// TIA Portal project "Trabajo" (V15)

(* hardware
DEVICE "S7-1200 station_1"  S7-1200 Station
   slot 0: "Rack_0"  S7-1200 Rack  Rack  V1.0
   slot 1: "PLC_1"  CPU 1215C AC/DC/Rly  6ES7 215-1BG40-0XB0  V4.2
*)

// ===== PLC "PLC_1"  CPU 1215C AC/DC/Rly =====

VAR_GLOBAL   // PLC tag table "Tabla de variables estándar"
   "Marcha" AT %I0.0 : Bool;
   "STOP" AT %I0.1 : Bool;
   "Automático" AT %I0.2 : Bool;
   "C1 Extendido" AT %I0.3 : Bool;
   "C1 Recogido" AT %I0.4 : Bool;
   "C2 Extendido" AT %I0.5 : Bool;
   "C2 Recogido" AT %I0.6 : Bool;
   "C3 Extendido" AT %I0.7 : Bool;
   "C3 Recogido" AT %I1.0 : Bool;
   "Alimentación" AT %I1.1 : Bool;
   "Pieza Mesa" AT %I1.2 : Bool;
   "Marcha 0" AT %M30.0 : Bool;
   "Marcha 1" AT %M30.1 : Bool;
   "Marcha 2" AT %M30.2 : Bool;
   "Marcha 3" AT %M30.3 : Bool;
   "Marcha 4" AT %M30.4 : Bool;
   "Marcha 5" AT %M30.5 : Bool;
   "Marcha 6" AT %M30.6 : Bool;
   "Marcha 7" AT %M30.7 : Bool;
   "Marcha 8" AT %M31.0 : Bool;
   "Marcha 9" AT %M31.1 : Bool;
   "Marcha 10" AT %M31.2 : Bool;
   "Marcha 11" AT %M31.3 : Bool;
   "Marcha 12" AT %M31.4 : Bool;
   "STOP 0" AT %M3.0 : Bool;
   "STOP 1" AT %M3.1 : Bool;
   "STOP 2" AT %M3.2 : Bool;
   "STOP 3" AT %M3.3 : Bool;
   "STOP 4" AT %M3.4 : Bool;
   "STOP 5" AT %M3.5 : Bool;
   "C1 SET" AT %Q0.0 : Bool;
   "C1 RESET" AT %Q0.1 : Bool;
   "C2 SET" AT %Q0.2 : Bool;
   "C2 RESET" AT %Q0.3 : Bool;
   "C3 SET" AT %Q0.4 : Bool;
   "Cinta ON" AT %Q0.5 : Bool;
   "Cinta INVERSA" AT %Q0.6 : Bool;
   "NumPiezas" AT %MW50 : Int;
   "Marcha 13" AT %M31.5 : Bool;
   "Marcha 14" AT %M31.6 : Bool;
   "Tag_2" AT %MB3 : Byte;
   "Tag_3" AT %MW30 : Int;
   "Tag_1" AT %MW100 : Int;
END_VAR

// folder: System blocks/Program resources

DATA_BLOCK "T1"   // DB1
{ S7_Optimized_Access := 'TRUE' }
AUTHOR : Simatic
FAMILY : IEC
NAME : IEC_TMR
VERSION : 1.0
// stored: InstanceOfName IEC_TIMER
"IEC_TIMER"
BEGIN
END_DATA_BLOCK

DATA_BLOCK "T2"   // DB2
{ S7_Optimized_Access := 'TRUE' }
AUTHOR : Simatic
FAMILY : IEC
NAME : IEC_TMR
VERSION : 1.0
// stored: InstanceOfName IEC_TIMER
"IEC_TIMER"
BEGIN
END_DATA_BLOCK

DATA_BLOCK "T3"   // DB3
{ S7_Optimized_Access := 'TRUE' }
AUTHOR : Simatic
FAMILY : IEC
NAME : IEC_TMR
VERSION : 1.0
// stored: InstanceOfName IEC_TIMER
"IEC_TIMER"
BEGIN
END_DATA_BLOCK

DATA_BLOCK "Contador"   // DB4
{ S7_Optimized_Access := 'TRUE' }
AUTHOR : Simatic
FAMILY : IEC
NAME : CNTR
VERSION : 1.0
// stored: InstanceOfName IEC_COUNTER
"IEC_COUNTER"
BEGIN
END_DATA_BLOCK

// folder: (top level)

FUNCTION "F_Marcha" : Void   // FC1, LAD
{ S7_Optimized_Access := 'TRUE' }
VERSION : 0.1
BEGIN

REGION Network 1: Etapa 0
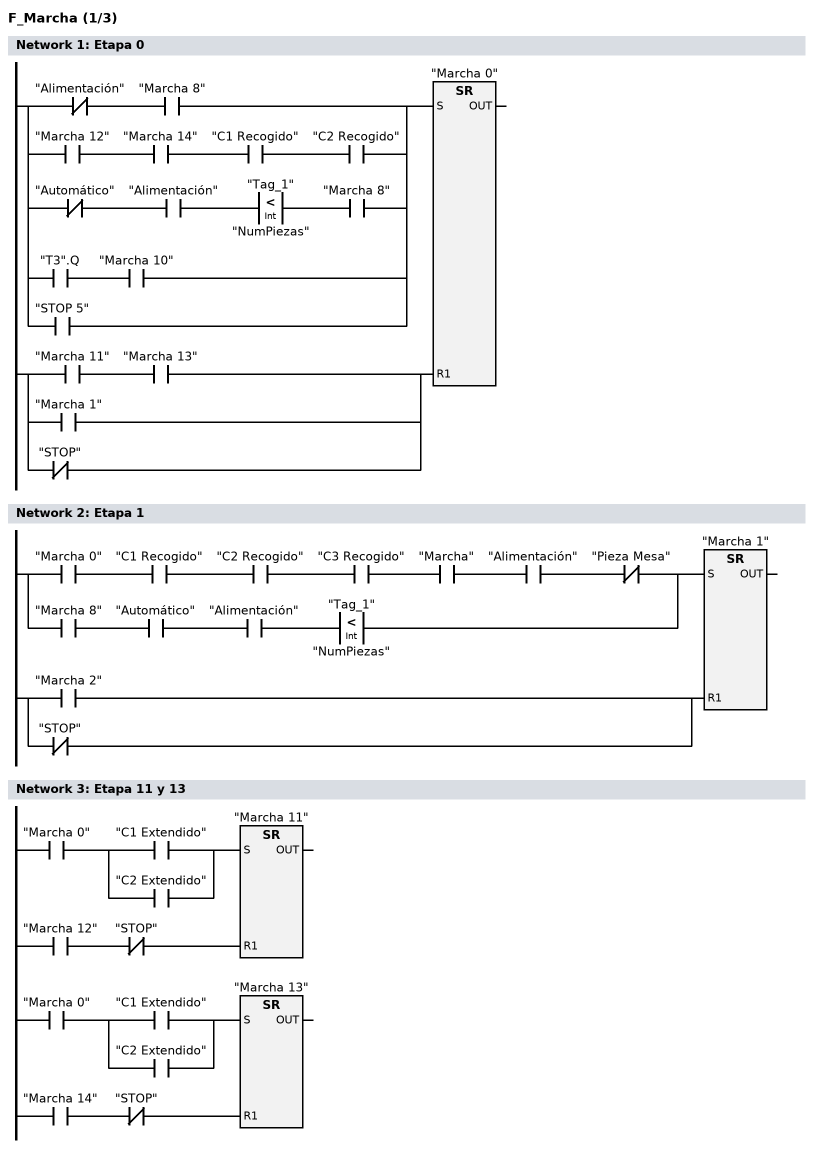
   RUNG wire#powerrail
      I_Contact( "Alimentación" )
      Contact( "Marcha 8" )
      wire#w1
      S_SR(operand := "Marcha 0", r1 := wire#w2)
   END_RUNG
   RUNG wire#powerrail
      Contact( "Marcha 12" )
      Contact( "Marcha 14" )
      Contact( "C1 Recogido" )
      Contact( "C2 Recogido" )
   END_RUNG wire#w1
   RUNG wire#powerrail
      I_Contact( "Automático" )
      Contact( "Alimentación" )
      { S7_Templates := "SrcType := Int" } LT_Contact(in1 := "Tag_1", in2 := "NumPiezas")
      Contact( "Marcha 8" )
   END_RUNG wire#w1
   RUNG wire#powerrail
      Contact( "T3".Q )
      Contact( "Marcha 10" )
   END_RUNG wire#w1
   RUNG wire#powerrail
      Contact( "STOP 5" )
   END_RUNG wire#w1
   RUNG wire#powerrail
      Contact( "Marcha 11" )
      Contact( "Marcha 13" )
   END_RUNG wire#w2
   RUNG wire#powerrail
      Contact( "Marcha 1" )
   END_RUNG wire#w2
   RUNG wire#powerrail
      I_Contact( "STOP" )
   END_RUNG wire#w2
   // the same network as SCL:
   IF (NOT "Alimentación" AND "Marcha 8") OR ("Marcha 12" AND "Marcha 14" AND "C1 Recogido" AND "C2 Recogido") OR (NOT "Automático" AND "Alimentación" AND ("Tag_1" < "NumPiezas") AND "Marcha 8") OR ("T3".Q AND "Marcha 10") OR "STOP 5" THEN
       "Marcha 0" := TRUE;   // SR flip-flop
   END_IF;
   IF ("Marcha 11" AND "Marcha 13") OR "Marcha 1" OR NOT "STOP" THEN "Marcha 0" := FALSE; END_IF;
END_REGION

REGION Network 2: Etapa 1
   RUNG wire#powerrail
      Contact( "Marcha 0" )
      Contact( "C1 Recogido" )
      Contact( "C2 Recogido" )
      Contact( "C3 Recogido" )
      Contact( "Marcha" )
      Contact( "Alimentación" )
      I_Contact( "Pieza Mesa" )
      wire#w1
      S_SR(operand := "Marcha 1", r1 := wire#w2)
   END_RUNG
   RUNG wire#powerrail
      Contact( "Marcha 8" )
      Contact( "Automático" )
      Contact( "Alimentación" )
      { S7_Templates := "SrcType := Int" } LT_Contact(in1 := "Tag_1", in2 := "NumPiezas")
   END_RUNG wire#w1
   RUNG wire#powerrail
      Contact( "Marcha 2" )
   END_RUNG wire#w2
   RUNG wire#powerrail
      I_Contact( "STOP" )
   END_RUNG wire#w2
   // the same network as SCL:
   IF ("Marcha 0" AND "C1 Recogido" AND "C2 Recogido" AND "C3 Recogido" AND "Marcha" AND "Alimentación" AND NOT "Pieza Mesa") OR ("Marcha 8" AND "Automático" AND "Alimentación" AND ("Tag_1" < "NumPiezas")) THEN
       "Marcha 1" := TRUE;   // SR flip-flop
   END_IF;
   IF "Marcha 2" OR NOT "STOP" THEN "Marcha 1" := FALSE; END_IF;
END_REGION

REGION Network 3: Etapa 11 y 13
   RUNG wire#powerrail
      Contact( "Marcha 0" )
      wire#w1
      Contact( "C1 Extendido" )
      wire#w2
      S_SR(operand := "Marcha 11", r1 := wire#w3)
   END_RUNG
   RUNG wire#w1
      Contact( "C2 Extendido" )
   END_RUNG wire#w2
   RUNG wire#powerrail
      Contact( "Marcha 12" )
      I_Contact( "STOP" )
   END_RUNG wire#w3
   RUNG wire#powerrail
      Contact( "Marcha 0" )
      wire#w4
      Contact( "C1 Extendido" )
      wire#w5
      S_SR(operand := "Marcha 13", r1 := wire#w6)
   END_RUNG
   RUNG wire#w4
      Contact( "C2 Extendido" )
   END_RUNG wire#w5
   RUNG wire#powerrail
      Contact( "Marcha 14" )
      I_Contact( "STOP" )
   END_RUNG wire#w6
   // the same network as SCL:
   IF "Marcha 0" AND ("C1 Extendido" OR "C2 Extendido") THEN
       "Marcha 11" := TRUE;   // SR flip-flop
   END_IF;
   IF "Marcha 12" AND NOT "STOP" THEN "Marcha 11" := FALSE; END_IF;
   IF "Marcha 0" AND ("C1 Extendido" OR "C2 Extendido") THEN
       "Marcha 13" := TRUE;   // SR flip-flop
   END_IF;
   IF "Marcha 14" AND NOT "STOP" THEN "Marcha 13" := FALSE; END_IF;
END_REGION

REGION Network 4: Etapa 12 y 14
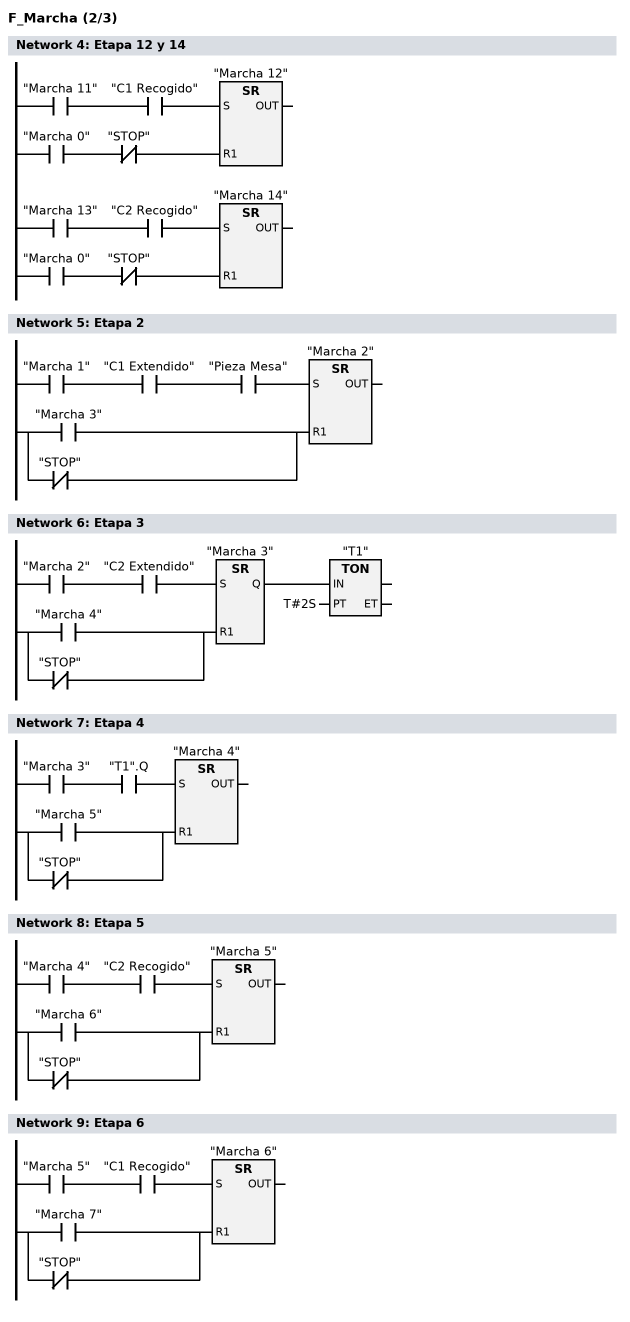
   RUNG wire#powerrail
      Contact( "Marcha 11" )
      Contact( "C1 Recogido" )
      S_SR(operand := "Marcha 12", r1 := wire#w1)
   END_RUNG
   RUNG wire#powerrail
      Contact( "Marcha 0" )
      I_Contact( "STOP" )
   END_RUNG wire#w1
   RUNG wire#powerrail
      Contact( "Marcha 13" )
      Contact( "C2 Recogido" )
      S_SR(operand := "Marcha 14", r1 := wire#w2)
   END_RUNG
   RUNG wire#powerrail
      Contact( "Marcha 0" )
      I_Contact( "STOP" )
   END_RUNG wire#w2
   // the same network as SCL:
   IF "Marcha 11" AND "C1 Recogido" THEN
       "Marcha 12" := TRUE;   // SR flip-flop
   END_IF;
   IF "Marcha 0" AND NOT "STOP" THEN "Marcha 12" := FALSE; END_IF;
   IF "Marcha 13" AND "C2 Recogido" THEN
       "Marcha 14" := TRUE;   // SR flip-flop
   END_IF;
   IF "Marcha 0" AND NOT "STOP" THEN "Marcha 14" := FALSE; END_IF;
END_REGION

REGION Network 5: Etapa 2
   RUNG wire#powerrail
      Contact( "Marcha 1" )
      Contact( "C1 Extendido" )
      Contact( "Pieza Mesa" )
      S_SR(operand := "Marcha 2", r1 := wire#w1)
   END_RUNG
   RUNG wire#powerrail
      Contact( "Marcha 3" )
   END_RUNG wire#w1
   RUNG wire#powerrail
      I_Contact( "STOP" )
   END_RUNG wire#w1
   // the same network as SCL:
   IF "Marcha 1" AND "C1 Extendido" AND "Pieza Mesa" THEN
       "Marcha 2" := TRUE;   // SR flip-flop
   END_IF;
   IF "Marcha 3" OR NOT "STOP" THEN "Marcha 2" := FALSE; END_IF;
END_REGION

REGION Network 6: Etapa 3
   IF "Marcha 2" AND "C2 Extendido" THEN
       "Marcha 3" := TRUE;   // SR flip-flop
   END_IF;
   IF "Marcha 4" OR NOT "STOP" THEN "Marcha 3" := FALSE; END_IF;
   "T1".TON(IN := "Marcha 3", PT := T#2S);
END_REGION

REGION Network 7: Etapa 4
   RUNG wire#powerrail
      Contact( "Marcha 3" )
      Contact( "T1".Q )
      S_SR(operand := "Marcha 4", r1 := wire#w1)
   END_RUNG
   RUNG wire#powerrail
      Contact( "Marcha 5" )
   END_RUNG wire#w1
   RUNG wire#powerrail
      I_Contact( "STOP" )
   END_RUNG wire#w1
   // the same network as SCL:
   IF "Marcha 3" AND "T1".Q THEN
       "Marcha 4" := TRUE;   // SR flip-flop
   END_IF;
   IF "Marcha 5" OR NOT "STOP" THEN "Marcha 4" := FALSE; END_IF;
END_REGION

REGION Network 8: Etapa 5
   RUNG wire#powerrail
      Contact( "Marcha 4" )
      Contact( "C2 Recogido" )
      S_SR(operand := "Marcha 5", r1 := wire#w1)
   END_RUNG
   RUNG wire#powerrail
      Contact( "Marcha 6" )
   END_RUNG wire#w1
   RUNG wire#powerrail
      I_Contact( "STOP" )
   END_RUNG wire#w1
   // the same network as SCL:
   IF "Marcha 4" AND "C2 Recogido" THEN
       "Marcha 5" := TRUE;   // SR flip-flop
   END_IF;
   IF "Marcha 6" OR NOT "STOP" THEN "Marcha 5" := FALSE; END_IF;
END_REGION

REGION Network 9: Etapa 6
   RUNG wire#powerrail
      Contact( "Marcha 5" )
      Contact( "C1 Recogido" )
      S_SR(operand := "Marcha 6", r1 := wire#w1)
   END_RUNG
   RUNG wire#powerrail
      Contact( "Marcha 7" )
   END_RUNG wire#w1
   RUNG wire#powerrail
      I_Contact( "STOP" )
   END_RUNG wire#w1
   // the same network as SCL:
   IF "Marcha 5" AND "C1 Recogido" THEN
       "Marcha 6" := TRUE;   // SR flip-flop
   END_IF;
   IF "Marcha 7" OR NOT "STOP" THEN "Marcha 6" := FALSE; END_IF;
END_REGION

REGION Network 10: Etapa 7
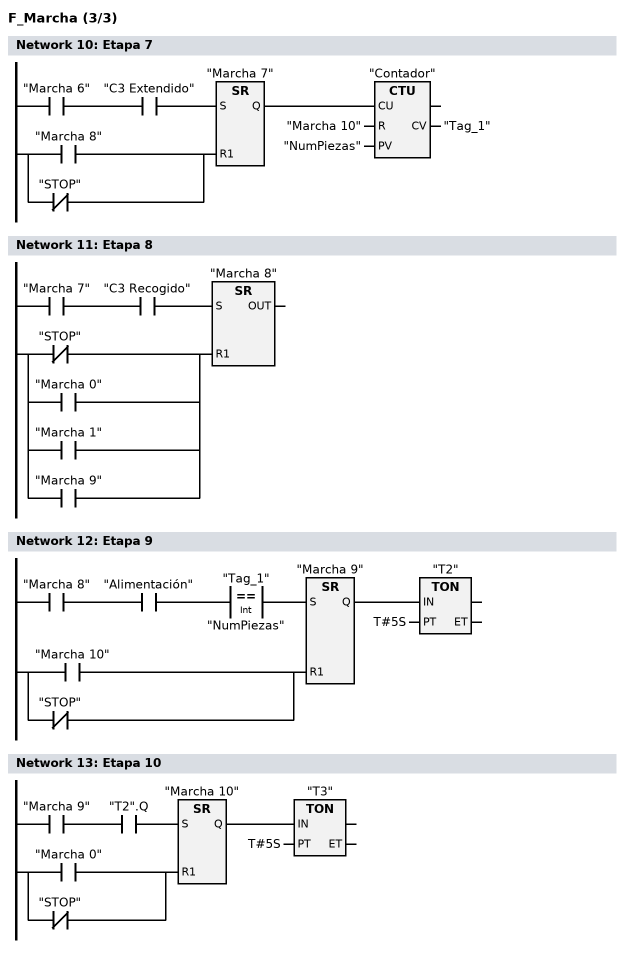
   IF "Marcha 6" AND "C3 Extendido" THEN
       "Marcha 7" := TRUE;   // SR flip-flop
   END_IF;
   IF "Marcha 8" OR NOT "STOP" THEN "Marcha 7" := FALSE; END_IF;
   "Contador".CTU(CU := "Marcha 7", R := "Marcha 10", PV := "NumPiezas", CV => "Tag_1");
END_REGION

REGION Network 11: Etapa 8
   RUNG wire#powerrail
      Contact( "Marcha 7" )
      Contact( "C3 Recogido" )
      S_SR(operand := "Marcha 8", r1 := wire#w1)
   END_RUNG
   RUNG wire#powerrail
      I_Contact( "STOP" )
   END_RUNG wire#w1
   RUNG wire#powerrail
      Contact( "Marcha 0" )
   END_RUNG wire#w1
   RUNG wire#powerrail
      Contact( "Marcha 1" )
   END_RUNG wire#w1
   RUNG wire#powerrail
      Contact( "Marcha 9" )
   END_RUNG wire#w1
   // the same network as SCL:
   IF "Marcha 7" AND "C3 Recogido" THEN
       "Marcha 8" := TRUE;   // SR flip-flop
   END_IF;
   IF NOT "STOP" OR "Marcha 0" OR "Marcha 1" OR "Marcha 9" THEN "Marcha 8" := FALSE; END_IF;
END_REGION

REGION Network 12: Etapa 9
   IF "Marcha 8" AND "Alimentación" AND ("Tag_1" = "NumPiezas") THEN
       "Marcha 9" := TRUE;   // SR flip-flop
   END_IF;
   IF "Marcha 10" OR NOT "STOP" THEN "Marcha 9" := FALSE; END_IF;
   "T2".TON(IN := "Marcha 9", PT := T#5S);
END_REGION

REGION Network 13: Etapa 10
   IF "Marcha 9" AND "T2".Q THEN
       "Marcha 10" := TRUE;   // SR flip-flop
   END_IF;
   IF "Marcha 0" OR NOT "STOP" THEN "Marcha 10" := FALSE; END_IF;
   "T3".TON(IN := "Marcha 10", PT := T#5S);
END_REGION
END_FUNCTION

FUNCTION "F_STOP" : Void   // FC2, LAD
{ S7_Optimized_Access := 'TRUE' }
VERSION : 0.1
BEGIN

REGION Network 1: Etapa 0
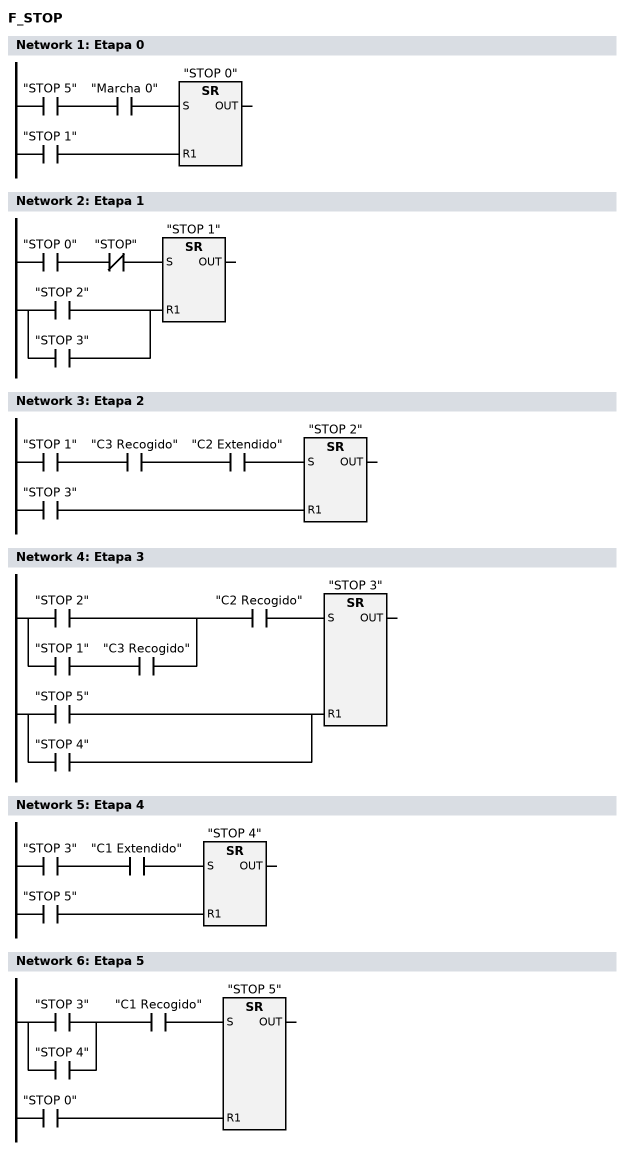
   RUNG wire#powerrail
      Contact( "STOP 5" )
      Contact( "Marcha 0" )
      S_SR(operand := "STOP 0", r1 := wire#w1)
   END_RUNG
   RUNG wire#powerrail
      Contact( "STOP 1" )
   END_RUNG wire#w1
   // the same network as SCL:
   IF "STOP 5" AND "Marcha 0" THEN
       "STOP 0" := TRUE;   // SR flip-flop
   END_IF;
   IF "STOP 1" THEN "STOP 0" := FALSE; END_IF;
END_REGION

REGION Network 2: Etapa 1
   RUNG wire#powerrail
      Contact( "STOP 0" )
      I_Contact( "STOP" )
      S_SR(operand := "STOP 1", r1 := wire#w1)
   END_RUNG
   RUNG wire#powerrail
      Contact( "STOP 2" )
   END_RUNG wire#w1
   RUNG wire#powerrail
      Contact( "STOP 3" )
   END_RUNG wire#w1
   // the same network as SCL:
   IF "STOP 0" AND NOT "STOP" THEN
       "STOP 1" := TRUE;   // SR flip-flop
   END_IF;
   IF "STOP 2" OR "STOP 3" THEN "STOP 1" := FALSE; END_IF;
END_REGION

REGION Network 3: Etapa 2
   RUNG wire#powerrail
      Contact( "STOP 1" )
      Contact( "C3 Recogido" )
      Contact( "C2 Extendido" )
      S_SR(operand := "STOP 2", r1 := wire#w1)
   END_RUNG
   RUNG wire#powerrail
      Contact( "STOP 3" )
   END_RUNG wire#w1
   // the same network as SCL:
   IF "STOP 1" AND "C3 Recogido" AND "C2 Extendido" THEN
       "STOP 2" := TRUE;   // SR flip-flop
   END_IF;
   IF "STOP 3" THEN "STOP 2" := FALSE; END_IF;
END_REGION

REGION Network 4: Etapa 3
   RUNG wire#powerrail
      Contact( "STOP 2" )
      wire#w1
      Contact( "C2 Recogido" )
      S_SR(operand := "STOP 3", r1 := wire#w2)
   END_RUNG
   RUNG wire#powerrail
      Contact( "STOP 1" )
      Contact( "C3 Recogido" )
   END_RUNG wire#w1
   RUNG wire#powerrail
      Contact( "STOP 5" )
   END_RUNG wire#w2
   RUNG wire#powerrail
      Contact( "STOP 4" )
   END_RUNG wire#w2
   // the same network as SCL:
   IF ("STOP 2" OR ("STOP 1" AND "C3 Recogido")) AND "C2 Recogido" THEN
       "STOP 3" := TRUE;   // SR flip-flop
   END_IF;
   IF "STOP 5" OR "STOP 4" THEN "STOP 3" := FALSE; END_IF;
END_REGION

REGION Network 5: Etapa 4
   RUNG wire#powerrail
      Contact( "STOP 3" )
      Contact( "C1 Extendido" )
      S_SR(operand := "STOP 4", r1 := wire#w1)
   END_RUNG
   RUNG wire#powerrail
      Contact( "STOP 5" )
   END_RUNG wire#w1
   // the same network as SCL:
   IF "STOP 3" AND "C1 Extendido" THEN
       "STOP 4" := TRUE;   // SR flip-flop
   END_IF;
   IF "STOP 5" THEN "STOP 4" := FALSE; END_IF;
END_REGION

REGION Network 6: Etapa 5
   RUNG wire#powerrail
      Contact( "STOP 3" )
      wire#w1
      Contact( "C1 Recogido" )
      S_SR(operand := "STOP 5", r1 := wire#w2)
   END_RUNG
   RUNG wire#powerrail
      Contact( "STOP 4" )
   END_RUNG wire#w1
   RUNG wire#powerrail
      Contact( "STOP 0" )
   END_RUNG wire#w2
   // the same network as SCL:
   IF ("STOP 3" OR "STOP 4") AND "C1 Recogido" THEN
       "STOP 5" := TRUE;   // SR flip-flop
   END_IF;
   IF "STOP 0" THEN "STOP 5" := FALSE; END_IF;
END_REGION
END_FUNCTION

FUNCTION "Salidas" : Void   // FC3, LAD
{ S7_Optimized_Access := 'TRUE' }
VERSION : 0.1
BEGIN

REGION Network 1: Set Cilindro 1
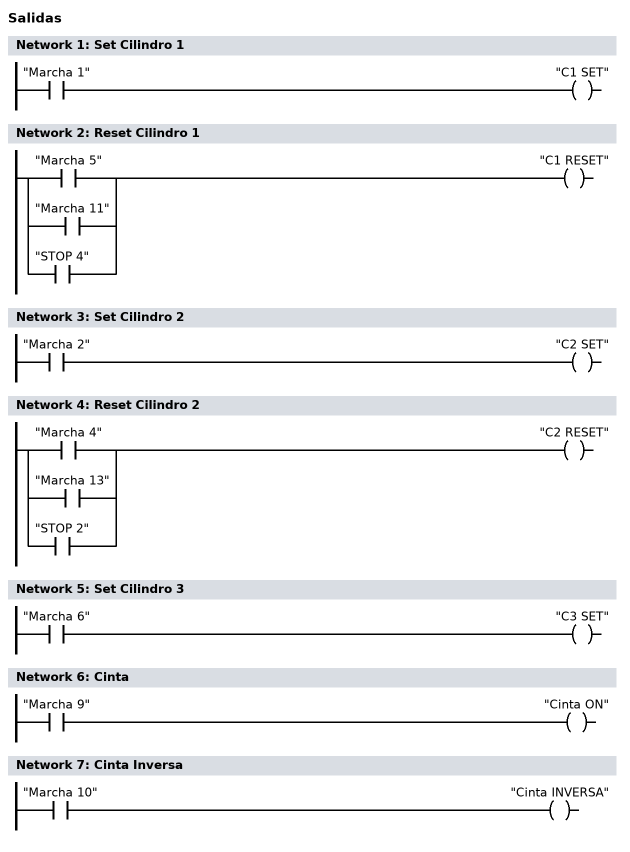
   RUNG wire#powerrail
      Contact( "Marcha 1" )
      Coil( "C1 SET" )
   END_RUNG
   // the same network as SCL:
   "C1 SET" := "Marcha 1";
END_REGION

REGION Network 2: Reset Cilindro 1
   RUNG wire#powerrail
      Contact( "Marcha 5" )
      wire#w1
      Coil( "C1 RESET" )
   END_RUNG
   RUNG wire#powerrail
      Contact( "Marcha 11" )
   END_RUNG wire#w1
   RUNG wire#powerrail
      Contact( "STOP 4" )
   END_RUNG wire#w1
   // the same network as SCL:
   "C1 RESET" := "Marcha 5" OR "Marcha 11" OR "STOP 4";
END_REGION

REGION Network 3: Set Cilindro 2
   RUNG wire#powerrail
      Contact( "Marcha 2" )
      Coil( "C2 SET" )
   END_RUNG
   // the same network as SCL:
   "C2 SET" := "Marcha 2";
END_REGION

REGION Network 4: Reset Cilindro 2
   RUNG wire#powerrail
      Contact( "Marcha 4" )
      wire#w1
      Coil( "C2 RESET" )
   END_RUNG
   RUNG wire#powerrail
      Contact( "Marcha 13" )
   END_RUNG wire#w1
   RUNG wire#powerrail
      Contact( "STOP 2" )
   END_RUNG wire#w1
   // the same network as SCL:
   "C2 RESET" := "Marcha 4" OR "Marcha 13" OR "STOP 2";
END_REGION

REGION Network 5: Set Cilindro 3
   RUNG wire#powerrail
      Contact( "Marcha 6" )
      Coil( "C3 SET" )
   END_RUNG
   // the same network as SCL:
   "C3 SET" := "Marcha 6";
END_REGION

REGION Network 6: Cinta
   RUNG wire#powerrail
      Contact( "Marcha 9" )
      Coil( "Cinta ON" )
   END_RUNG
   // the same network as SCL:
   "Cinta ON" := "Marcha 9";
END_REGION

REGION Network 7: Cinta Inversa
   RUNG wire#powerrail
      Contact( "Marcha 10" )
      Coil( "Cinta INVERSA" )
   END_RUNG
   // the same network as SCL:
   "Cinta INVERSA" := "Marcha 10";
END_REGION
END_FUNCTION

ORGANIZATION_BLOCK "Main"   // OB1, LAD, ProgramCycle
TITLE = "Main Program Sweep (Cycle)"
{ S7_Optimized_Access := 'TRUE' }
VERSION : 0.1
// Main con funciones de marcha, STOP y salidas.
   VAR_INPUT
      Initial_Call : Bool;   // Initial call of this OB
      Remanence : Bool;   // =True, if remanent data are available
   END_VAR
BEGIN

REGION Network 1: Función Marcha
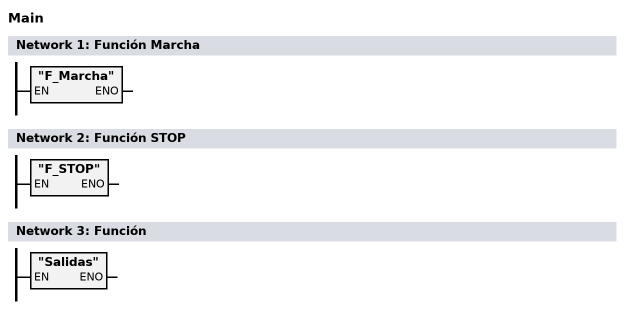
   RUNG wire#powerrail
      "F_Marcha"()
   END_RUNG
   // the same network as SCL:
   "F_Marcha"();
END_REGION

REGION Network 2: Función STOP
   RUNG wire#powerrail
      "F_STOP"()
   END_RUNG
   // the same network as SCL:
   "F_STOP"();
END_REGION

REGION Network 3: Función
   RUNG wire#powerrail
      "Salidas"()
   END_RUNG
   // the same network as SCL:
   "Salidas"();
END_REGION
END_ORGANIZATION_BLOCK

ORGANIZATION_BLOCK "Startup"   // OB100, LAD, Startup
TITLE = "Complete Restart" / Start up Marcha y STOP
{ S7_Optimized_Access := 'TRUE' }
VERSION : 0.1
   VAR_INPUT
      LostRetentive : Bool;   // True if retentive data are lost
      LostRTC : Bool;   // True if date and time are lost
   END_VAR
BEGIN

REGION Network 1
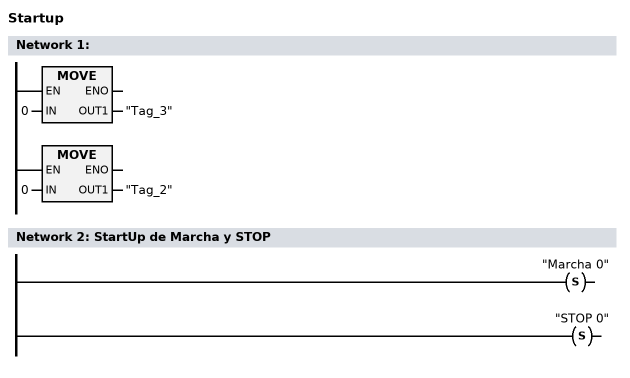
   RUNG wire#powerrail
      Move(in := 0, out1 => "Tag_3")
   END_RUNG
   RUNG wire#powerrail
      Move(in := 0, out1 => "Tag_2")
   END_RUNG
   // the same network as SCL:
   "Tag_3" := 0;
   "Tag_2" := 0;
END_REGION

REGION Network 2: StartUp de Marcha y STOP
   RUNG wire#powerrail
      S_Coil( "Marcha 0" )
   END_RUNG
   RUNG wire#powerrail
      S_Coil( "STOP 0" )
   END_RUNG
   // the same network as SCL:
   "Marcha 0" := TRUE;
   "STOP 0" := TRUE;
END_REGION
END_ORGANIZATION_BLOCK